TYPE M2YAxisStatuses :
STRUCT
	///Is the axis healthy?
	healthStatus: HealthStatus;
END_STRUCT
END_TYPE

(* stored: Version 1.1.0.1, ProductVersion 3.1.4019.2
   DUT M2YAxisStatuses: Id {09c6578d-d389-4ff4-859f-310af4857145} *)
